FUNCTION_BLOCK "MES_CHeck"
VAR
  Station_1 : "MES Check_fb";
  Station_2 : "MES Check_fb";
  Station_3 : "MES Check_fb";
  Station_4 : "MES Check_fb";
  Station_5 : "MES Check_fb";
  Station_6 : "MES Check_fb";
  Station_7 : "MES Check_fb";
  Station_8 : "MES Check_fb";
END_VAR
BEGIN
  // Původní jazyk: LAD
  // Zdroj XML: EXPORT/Program blocks/OP010/11_MES/MES_CHeck.xml
  // (Žádný StructuredText network nebyl nalezen; LAD/STL/GRAPH není automaticky překládán.)
END_FUNCTION_BLOCK
